// TIA Portal V20 export
DATA_BLOCK "DB_AxisPosition"   // DB411
// stored: AutoNumber false, InstanceOfName FB_AxisPosition, InstanceOfType FB
"FB_AxisPosition"
   // VAR
   //    sError { ExternalAccessible := 'False'; ExternalVisible := 'False'; ExternalWritable := 'False'} : Bool;
   //    sNDR { ExternalAccessible := 'False'; ExternalVisible := 'False'; ExternalWritable := 'False'} : Bool;
   //    sState { ExternalAccessible := 'False'; ExternalVisible := 'False'; ExternalWritable := 'False'} : Word;
   //    sAxis01_X : Struct
   //       "$AA_IM" : LReal;
   //       "$MA_POS_LIMIT_MINUS" : LReal;
   //       "$MA_POS_LIMIT_MINUS2" : LReal;
   //       "$MA_POS_LIMIT_PLUS" : LReal;
   //       "$MA_POS_LIMIT_PLUS2" : LReal;
   //       "$MA_JOG_VELO" : LReal;
   //       "$MA_JOG_VELO_RAPID" : LReal;
   //       "$MA_MAX_AX_VELO" : LReal;
   //       "$A1_M_FP_POS4_30600" : LReal;
   //    END_STRUCT;
   //    sAxis02_Y : Struct
   //       "$AA_IM" : LReal;
   //       "$MA_POS_LIMIT_MINUS" : LReal;
   //       "$MA_POS_LIMIT_MINUS2" : LReal;
   //       "$MA_POS_LIMIT_PLUS" : LReal;
   //       "$MA_POS_LIMIT_PLUS2" : LReal;
   //       "$MA_JOG_VELO" : LReal;
   //       "$MA_JOG_VELO_RAPID" : LReal;
   //       "$MA_MAX_AX_VELO" : LReal;
   //    END_STRUCT;
   //    sAxis03_ZM : Struct
   //       "$AA_IM" : LReal;
   //       "$MA_POS_LIMIT_MINUS" : LReal;
   //       "$MA_POS_LIMIT_MINUS2" : LReal;
   //       "$MA_POS_LIMIT_PLUS" : LReal;
   //       "$MA_POS_LIMIT_PLUS2" : LReal;
   //       "$MA_JOG_VELO" : LReal;
   //       "$MA_JOG_VELO_RAPID" : LReal;
   //       "$MA_MAX_AX_VELO" : LReal;
   //    END_STRUCT;
   //    sAxis04_B : Struct
   //       "$AA_IM" : LReal;
   //       "$MA_POS_LIMIT_MINUS" : LReal;
   //       "$MA_POS_LIMIT_MINUS2" : LReal;
   //       "$MA_POS_LIMIT_PLUS" : LReal;
   //       "$MA_POS_LIMIT_PLUS2" : LReal;
   //       "$MA_JOG_VELO" : LReal;
   //       "$MA_JOG_VELO_RAPID" : LReal;
   //       "$MA_MAX_AX_VELO" : LReal;
   //    END_STRUCT;
   //    sAxis05_U1 : Struct
   //       "$AA_IM" : LReal;
   //       "$MA_POS_LIMIT_MINUS" : LReal;
   //       "$MA_POS_LIMIT_MINUS2" : LReal;
   //       "$MA_POS_LIMIT_PLUS" : LReal;
   //       "$MA_POS_LIMIT_PLUS2" : LReal;
   //       "$MA_JOG_VELO" : LReal;
   //       "$MA_JOG_VELO_RAPID" : LReal;
   //       "$MA_MAX_AX_VELO" : LReal;
   //    END_STRUCT;
   //    sAxis06_U2 : Struct
   //       "$AA_IM" : LReal;
   //       "$MA_POS_LIMIT_MINUS" : LReal;
   //       "$MA_POS_LIMIT_MINUS2" : LReal;
   //       "$MA_POS_LIMIT_PLUS" : LReal;
   //       "$MA_POS_LIMIT_PLUS2" : LReal;
   //       "$MA_JOG_VELO" : LReal;
   //       "$MA_JOG_VELO_RAPID" : LReal;
   //       "$MA_MAX_AX_VELO" : LReal;
   //       "$A1_M_FP_POS2_30600" : LReal;
   //    END_STRUCT;
   //    sAxis07_V : Struct
   //       "$AA_IM" : LReal;
   //       "$MA_POS_LIMIT_MINUS" : LReal;
   //       "$MA_POS_LIMIT_MINUS2" : LReal;
   //       "$MA_POS_LIMIT_PLUS" : LReal;
   //       "$MA_POS_LIMIT_PLUS2" : LReal;
   //       "$MA_JOG_VELO" : LReal;
   //       "$MA_JOG_VELO_RAPID" : LReal;
   //       "$MA_MAX_AX_VELO" : LReal;
   //    END_STRUCT;
   //    sAxis08_W : Struct
   //       "$AA_IM" : LReal;
   //       "$MA_POS_LIMIT_MINUS" : LReal;
   //       "$MA_POS_LIMIT_MINUS2" : LReal;
   //       "$MA_POS_LIMIT_PLUS" : LReal;
   //       "$MA_POS_LIMIT_PLUS2" : LReal;
   //       "$MA_JOG_VELO" : LReal;
   //       "$MA_JOG_VELO_RAPID" : LReal;
   //       "$MA_MAX_AX_VELO" : LReal;
   //    END_STRUCT;
   //    sAxis09_ZL : Struct
   //       "$AA_IM" : LReal;
   //       "$MA_POS_LIMIT_MINUS" : LReal;
   //       "$MA_POS_LIMIT_MINUS2" : LReal;
   //       "$MA_POS_LIMIT_PLUS" : LReal;
   //       "$MA_POS_LIMIT_PLUS2" : LReal;
   //       "$MA_JOG_VELO" : LReal;
   //       "$MA_JOG_VELO_RAPID" : LReal;
   //       "$MA_MAX_AX_VELO" : LReal;
   //    END_STRUCT;
   // END_VAR
BEGIN
END_DATA_BLOCK
